# EPICS SNL sequencer program: test/validate/pvGetCancel.st
/*************************************************************************\
Copyright (c) 2010-2012 Helmholtz-Zentrum Berlin f. Materialien
                        und Energie GmbH, Germany (HZB)
This file is distributed subject to a Software License Agreement found
in the file LICENSE that is included with this distribution.
\*************************************************************************/
program pvGetCancelTest

/* option +s; */

%%#include "../testSupport.h"

#define NRUNS 50

entry {
    seq_test_init(8*NRUNS);
    testDiag("start");
}

ss pvGetCancel {
    int x[2];
    int y[2] = {1,2};
    assign x to { "pvGetCancel1", "pvGetCancel2"};
    assign y to { "pvGetCancel1", "pvGetCancel2"};
    typename pvStat status;
    int n = 0;

    state done {
        when (n < NRUNS) {
            n++;
        } state test
        when (delay(0.2)) {
        } exit
    }
    state test {
        entry {
            testOk1(pvGet(x[0],ASYNC) == pvStatOK);
            testOk1(pvGet(x[1],ASYNC) == pvStatOK);
            pvGetCancel(x);
            x[0] = x[1] = 0;
            y[0] = y[1] = 1;
            testOk1(pvPut(y[0],SYNC) == pvStatOK);
            testOk1(pvPut(y[1],SYNC) == pvStatOK);
            testOk1(pvGet(x[0],ASYNC) == pvStatOK);
            testOk1(pvGet(x[1],ASYNC) == pvStatOK);
        }
        when (delay(5.0)) {
            testFail("pvGet completion timeout");
            testSkip(1,"further tests aborted");
        } exit
        when (pvGetComplete(x)) {
            testOk1(x[0] == y[0]);
            testOk1(x[1] == y[1]);
        } state done
    }
}

exit {
    testDiag("exit");
    seq_test_done();
}
